// TwinCAT 3 PLC project Test
// Title: Testlibrary
// Company: Eclipse Automation Penang
// Author: BC Yeoh
// ProjectVersion: 0.0.0.1
// Description: testing library
// ProgramVersion: 3.1.4024.0
// libraries:
//   Tc2_Standard, * (Beckhoff Automation GmbH)
//   Tc2_System, * (Beckhoff Automation GmbH)
//   Tc2_Utilities, * (Beckhoff Automation GmbH)
//   Tc3_Module, * (Beckhoff Automation GmbH)
// project tree:
//   DUTs/ E_EventType.TcDUT, ST_Event.TcDUT
//   / PlcTask.TcTTO
//   POUs/ Factorial.TcPOU, FB_EventBuffer.TcPOU, MAIN.TcPOU
//   Version/ Global_Version.TcGVL
// (motion and I/O tree: see PLC project 4 position demolding test system)
// real-time tasks:
//   TASK PlcTask: cycle T#10ms, priority 20, ADS port 350
//   TASK PlcTask1: cycle T#10ms, priority 21, ADS port 351
//   TASK PlcTask2: cycle T#10ms, priority 22, ADS port 352

CONFIGURATION Test
    RESOURCE PLC ON TwinCAT3
        TASK PlcTask(INTERVAL := T#10ms, PRIORITY := 22);
        PROGRAM MAIN WITH PlcTask : MAIN;
    END_RESOURCE
END_CONFIGURATION

// ---- DUTs/E_EventType.TcDUT
{attribute 'qualified_only'}
{attribute 'strict'}
{attribute 'to_string'}
TYPE E_EventType :
(
	Alarm := 0,
	Messages:=1,
	Warning:=2
);
END_TYPE

// ---- DUTs/ST_Event.TcDUT
TYPE ST_Event :
STRUCT
	eEventTypes: E_EventType;
	eEventSeverity: TcEventSeverity;
	eEventIdentity: UDINT;
	eEventText: STRING(255);
	dtTimestamp: DATE_AND_TIME;	
END_STRUCT
END_TYPE

// ---- Version/Global_Version.TcGVL
{attribute 'TcGenerated'}
{attribute 'no-analysis'}
{attribute 'linkalways'}
// This function has been automatically generated from the project information.
VAR_GLOBAL CONSTANT
	{attribute 'const_non_replaced'}
	stLibVersion_Testlibrary : ST_LibVersion := (iMajor := 0, iMinor := 0, iBuild := 0, iRevision := 1, nFlags := 0, sVersion := '0.0.0.1');
END_VAR

// ---- POUs/MAIN.TcPOU
PROGRAM MAIN
VAR
fbProfiler: Profiler;
stProfilerResult:PROFILERSTRUCT;
nAnsOfFactorial:ULINT;
END_VAR

fbProfiler(start:=TRUE,reset:=FALSE);
	Factorial(nAnsOfFactorial);	
fbProfiler(start:=FALSE);
stProfilerResult:= fbProfiler.DATA;

END_PROGRAM

// ---- POUs/Factorial.TcPOU
FUNCTION Factorial : ULINT
VAR_INPUT
	n:ULINT;
END_VAR
VAR
		nReturnValue:ULINT;
		i:ULINT;
END_VAR

nReturnValue:=1;
FOR i:=1 TO n BY 1 DO
	nReturnValue:= nReturnValue *i ;
END_FOR
Factorial:=nReturnValue;

END_FUNCTION

// ---- POUs/FB_EventBuffer.TcPOU
FUNCTION_BLOCK FB_EventBuffer

VAR
MemRingBuffer: FB_MemRingBuffer;	
aBufferArray  : ARRAY[0..Number_Of_Bytes_For_All_ST_Event] OF BYTE; (* Buffer memory used by FB_MemRingBuffer function block *)
END_VAR

VAR CONSTANT
	Size_Of_ST_Event: UDINT :=SIZEOF(ST_Event);
	Max_Number_Of_ST_Event: UDINT := 5;
	Number_Of_Bytes_For_All_ST_Event: UDINT := Size_Of_ST_Event*Max_Number_Of_ST_Event;
END_VAR

METHOD PUBLIC GetAndRemoveEvent
VAR_OUTPUT
	stEvent: ST_Event;
	bError : BOOL;
END_VAR
MemRingBuffer.A_RemoveHead(pRead:=ADR(stEvent),
						  	cbRead:=SIZEOF(stEvent),
							pBuffer:=ADR(aBufferArray),
							cbBuffer:=SIZEOF(aBufferArray));

bError:= NOT MemRingBuffer.bOk;
END_METHOD

METHOD PUBLIC TryToAddEvent
VAR_INPUT
	stEvent: REFERENCE TO ST_Event;
END_VAR

VAR_OUTPUT
    bError : BOOL;
END_VAR
MemRingBuffer.A_AddTail(pWrite:=ADR(stEvent),
						cbWrite:=SIZEOF(stEvent),
						pBuffer:=ADR(aBufferArray),cbBuffer:=SIZEOF(aBufferArray));
bError:= NOT MemRingBuffer.bOk;
END_METHOD

END_FUNCTION_BLOCK
